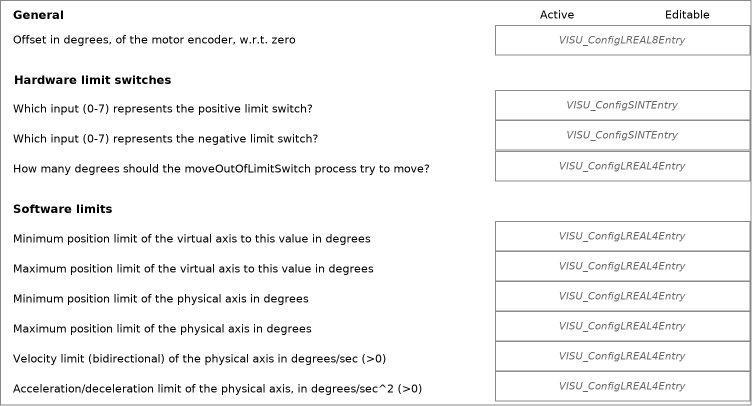
VISUALIZATION VISU_AxesConfig_Rotation_1  // 752x406
VAR_IN_OUT
    active : AxesRotationConfig;
    editable : AxesRotationConfig;
END_VAR
    Label (495,5 125x20), "Active"
    Label (625,5 125x20), "Editable"
    Label (10,25 360x30), "Offset in degrees, of the motor encoder, w.r.t. zero"
    Frame (495,25 255x30)
        shows VISU_ConfigLREAL8Entry(active := active.motorEncoderOffset, editable := editable.motorEncoderOffset)
    Label (10,94 475x30), "Which input (0-7) represents the positive limit switch?"
    Label (10,124 475x30), "Which input (0-7) represents the negative limit switch?"
    Label (10,154 475x30), "How many degrees should the moveOutOfLimitSwitch process try to move?"
    Label (11,65 150x30), "Hardware limit switches"
    Label (10,224 475x30), "Minimum position limit of the virtual axis to this value in degrees"
    Label (10,194 165x30), "Software limits"
    Label (10,254 475x30), "Maximum position limit of the virtual axis to this value in degrees"
    Label (10,284 475x30), "Minimum position limit of the physical axis in degrees"
    Label (10,314 475x30), "Maximum position limit of the physical axis in degrees"
    Label (10,344 475x30), "Velocity limit (bidirectional) of the physical axis in degrees/sec (>0)"
    Label (10,374 475x30), "Acceleration/deceleration limit of the physical axis, in degrees/sec^2 (>0)"
    Label (10,0 150x30), "General"
    Frame (495,90 255x30)
        shows VISU_ConfigSINTEntry(active := active.positiveLimitSwitchInput, editable := editable.positiveLimitSwitchInput)
    Frame (495,120 255x30)
        shows VISU_ConfigSINTEntry(active := active.negativeLimitSwitchInput, editable := editable.negativeLimitSwitchInput)
    Frame (495,151 255x30)
        shows VISU_ConfigLREAL4Entry(active := active.moveOutOfLimitSwitchDistance, editable := editable.moveOutOfLimitSwitchDistance)
    Frame (495,221 255x30)
        shows VISU_ConfigLREAL4Entry(active := active.minPositionLimitVirtualAxis, editable := editable.minPositionLimitVirtualAxis)
    Frame (495,251 255x30)
        shows VISU_ConfigLREAL4Entry(active := active.maxPositionLimitVirtualAxis, editable := editable.maxPositionLimitVirtualAxis)
    Frame (495,281 255x30)
        shows VISU_ConfigLREAL4Entry(active := active.minPositionLimitPhysicalAxis, editable := editable.minPositionLimitPhysicalAxis)
    Frame (495,311 255x30)
        shows VISU_ConfigLREAL4Entry(active := active.maxPositionLimitPhysicalAxis, editable := editable.maxPositionLimitPhysicalAxis)
    Frame (495,341 255x30)
        shows VISU_ConfigLREAL4Entry(active := active.velocityLimit, editable := editable.velocityLimit)
    Frame (495,371 255x30)
        shows VISU_ConfigLREAL4Entry(active := active.accelerationLimit, editable := editable.accelerationLimit)
END_VISUALIZATION

(* stored: Version 1.1.0.1, ProductVersion 3.1.4019.2
   Visu VISU_AxesConfig_Rotation_1: Id {17421c89-3998-4ee5-818d-c9ea21fceb8d} *)
